(* CODESYS project ers_co2_payload_decoder.library
   Company: PXL-Tech
   Title: ERS_CO2 Payload Decoder
   Placeholder: ERS_CO2 Payload Decoder
   Version: 1.0

Project tree, tasks and I/O mapping:
  libraries: Tc2_Standard, * (Beckhoff Automation GmbH); Tc2_System, * (Beckhoff Automation GmbH); Tc2_Utilities, * (Beckhoff Automation GmbH); Tc3_Module, * (Beckhoff Automation GmbH)
  DUTs/
  GVLs/
  POUs/
    function block ERS_CO2_PayloadDecoder [ST]
    program MAIN [ST]
  Version/
    global variables Global_Version
  VISUs/
*)

// Version/Global_Version
{attribute 'TcGenerated'}
// This function has been automatically generated from the project information.
VAR_GLOBAL CONSTANT
	{attribute 'const_non_replaced'}
	{attribute 'linkalways'}
	stLibVersion_ERS_CO2_Payload_Decoder : ST_LibVersion := (iMajor := 1, iMinor := 0, iBuild := 0, iRevision := 0, sVersion := '1.0');
END_VAR

// POUs/ERS_CO2_PayloadDecoder
FUNCTION_BLOCK ERS_CO2_PayloadDecoder
VAR_INPUT
	dataString 		: STRING(32);
END_VAR
VAR_OUTPUT
	Temperature 	: REAL;		//Temp -3276.8°C - 3276.7°C
	Humidity 		: BYTE;		//Humidity 0-100%
	X 				: REAL;		//Acceleration X -128 --> 127 +/-63 = 1G
	Y 				: REAL;		//Acceleration Y -128 --> 127 +/-63 = 1G
	Z 				: REAL;		//Acceleration Z -128 --> 127 +/-63 = 1G
	Light 			: WORD; 	//Light 0 - 65535 Lux
	Motion 			: BYTE;		//No of motion 0-255
	Co2				: WORD;		//Co2 0-65535 ppm 
	Vdd				: WORD;		//VDD 0-65535mV
	Analog1			: WORD;		//VDD 0-65535mV
	Lat				: DWORD;	//Latitude binary
	Lon				: DWORD;	//Longitude binary
	Pulse1			: WORD;		//Relative pulse count
	pulseAbs		: DWORD;	//no 0 - 0xFFFFFFFF
	ExternalTemp	: REAL;		//External temp -3276.5C-->3276.5C
	Digital			: BYTE;		//Value 1 or 0
	Distance		: WORD;		//Distance in mm
	AccMotion		: BYTE;		//Number of vibration/motion
	IrInternalTemp	: REAL;		//Internal temp -3276.5C - 3276.5C
	IrExternalTemp	: REAL;		//External temp -3276.5C - 3276.5C
	Occupancy		: BYTE;		//Data
	Waterleak		: BYTE;		//Data 0-255
	Pressure		: REAL;		//Pressure data(hPa)
	SoundPeak		: BYTE;		//Sound peak
	SoundAvg		: BYTE;		//Sound average
	Pulse2			: WORD;		//0 - 0xFFFF
	PulseAbs2		: DWORD;	//no 0 - 0xFFFFFFFF
	Analog2			: WORD;		//Voltage in mV
	ExternalTemp2	: REAL;		//External temp2 -3276.5C - 3276.5C
	
	msgIDs			: ARRAY[1..8] OF BYTE;
END_VAR
VAR
	dataBuf			: ARRAY[1..16] OF BYTE;
	i				: INT;
	j				: INT;
END_VAR
VAR CONSTANT
	ID_Temp			:	BYTE	:= 16#01;	//Temperature
	ID_Rh			:	BYTE	:= 16#02;	//Humidity
	ID_Acc			:	BYTE	:= 16#03;	//X, Y, Z
	ID_Light		:	BYTE	:= 16#04;	//Light
	ID_Motion		:	BYTE	:= 16#05;	//Motion
	ID_Co2			:	BYTE	:= 16#06;	//Co2
	ID_Vdd			:	BYTE	:= 16#07;	//Vdd
	ID_Analog1		:	BYTE	:= 16#08;	//Analog1
	ID_Gps			:	BYTE	:= 16#09;	//Lat, Lon
	ID_Pulse1		:	BYTE	:= 16#0A;	//Pulse1
	ID_Pulse1_Abs	:	BYTE	:= 16#0B;	//Pulse1_Abs
	ID_Ext_Temp1	:	BYTE	:= 16#0C;	//ExternalTemp
	ID_Ext_Digital	:	BYTE	:= 16#0D;	//Digital
	ID_Ext_distance	:	BYTE	:= 16#0E;	//Distance
	ID_Acc_Motion	:	BYTE	:= 16#0F;	//AccMotion
	ID_Ir_Temp		:	BYTE	:= 16#10;	//IrInternalTemp, IrExternalTemp
	ID_Occupancy	:	BYTE	:= 16#11;	//Occupancy
	ID_Waterleak	:	BYTE	:= 16#12;	//Waterleak
	ID_Grideye		:	BYTE	:= 16#13;
	ID_Pressure		:	BYTE	:= 16#14;	//Pressure
	ID_Sound		:	BYTE	:= 16#15;	//SoundPeak, SoundAvg
	ID_Pulse2		:	BYTE	:= 16#16;	//Pulse2
	ID_Pulse2_Abs	:	BYTE	:= 16#17;	//Pulse2_Abs
	ID_Analog2		:	BYTE	:= 16#18;	//Analog2
	ID_Ext_Temp2	:	BYTE	:= 16#19;	//ExternalTemp2
END_VAR

HEXSTR_TO_DATA(dataString, ADR(dataBuf), SIZEOF(dataBuf));

j := 1;
MEMSET(ADR(msgIDs), 0, SIZEOF(msgIDs));

FOR i := 1 TO 15 BY 1 DO;
	CASE dataBuf[i] OF
		ID_Temp:
			Temperature := WORD_TO_REAL(SHL(dataBuf[i + 1], 8) OR dataBuf[i + 2]) / 10;
			msgIDs[j] := ID_Temp;
			j := j + 1;
			i := i + 2;
		ID_Rh:
			Humidity := dataBuf[i + 1];
			msgIDs[j] := ID_Rh;
			j := j + 1;
			i := i + 1;
		ID_Acc:
			X := dataBuf[i + 1];
			Y := dataBuf[i + 2];
			Z := dataBuf[i + 3];
			msgIDs[j] := ID_Acc;
			j := j + 1;
			i := i + 3;
		ID_Light:
			Light := SHL(dataBuf[i + 1], 8) OR dataBuf[i + 2];
			msgIDs[j] := ID_Light;
			j := j + 1;
			i := i + 2;
		ID_Motion:
			Motion := dataBuf[i + 1];
			msgIDs[j] := ID_Motion;
			j := j + 1;
			i := i + 1;
		ID_Co2:
			Co2 := SHL(dataBuf[i + 1], 8) OR dataBuf[i + 2];
			msgIDs[j] := ID_Co2;
			j := j + 1;
			i := i + 2;
		ID_Vdd:
			Vdd := SHL(dataBuf[i + 1], 8) OR dataBuf[i + 2];
			msgIDs[j] := ID_Vdd;
			j := j + 1;
			i := i + 2;
		ID_Analog1:
			Analog1 := SHL(dataBuf[i + 1], 8) OR dataBuf[i + 2];
			msgIDs[j] := ID_Analog1;
			j := j + 1;
			i := i + 2;
		ID_Gps:
			Lat := SHL(dataBuf[i + 1], 16) OR SHL(dataBuf[i + 2], 8) OR dataBuf[i + 3];
			Lon := SHL(dataBuf[i + 4], 16) OR SHL(dataBuf[i + 5], 8) OR dataBuf[i + 6];
			msgIDs[j] := ID_Gps;
			j := j + 1;
			i := i + 6;
		ID_Pulse1:
			Pulse1 := SHL(dataBuf[i + 1], 8) OR dataBuf[i + 2];
			msgIDs[j] := ID_Pulse1;
			j := j + 1;
			i := i + 2;
		ID_Pulse1_Abs:
			PulseAbs := SHL(dataBuf[i + 1], 24) OR SHL(dataBuf[i + 2], 16) OR  SHL(dataBuf[i + 3], 8) OR dataBuf[i + 4];
			msgIDs[j] := ID_Pulse1_Abs;
			j := j + 1;
			i := i + 4;
		ID_Ext_Temp1:
			ExternalTemp := WORD_TO_REAL(SHL(dataBuf[i + 1], 8) OR dataBuf[i + 2]) / 10;
			msgIDs[j] := ID_Ext_Temp1;
			j := j + 1;
			i := i + 2;
		ID_Ext_Digital:
			Digital := dataBuf[i + 1];
			msgIDs[j] := ID_Ext_Digital;
			j := j + 1;
			i := i + 1;
		ID_Ext_distance:
			Distance := SHL(dataBuf[i + 1], 8) OR dataBuf[i + 2];
			msgIDs[j] := ID_Ext_distance;
			j := j + 1;
			i := i + 2;
		ID_Acc_Motion:
			AccMotion := dataBuf[i + 1];
			msgIDs[j] := ID_Acc_Motion;
			j := j + 1;
			i := i + 1;
		ID_Ir_Temp:
			IrInternalTemp := WORD_TO_REAL(SHL(dataBuf[i + 1], 8) OR dataBuf[i + 2]) / 10;
			IrExternalTemp := WORD_TO_REAL(SHL(dataBuf[i + 3], 8) OR dataBuf[i + 4]) / 10;
			msgIDs[j] := ID_Ir_Temp;
			j := j + 1;
			i := i + 4;
		ID_Occupancy:
			Occupancy := dataBuf[i + 1];
			msgIDs[j] := ID_Occupancy;
			j := j + 1;
			i := i + 1;
		ID_Waterleak:
			Waterleak := dataBuf[i + 1];
			msgIDs[j] := ID_Waterleak;
			j := j + 1;
			i := i + 1;
		ID_Grideye:
			msgIDs[j] := ID_Grideye;
			j := j + 1;
			i := i + 65;
		ID_Pressure:
			Pressure := DWORD_TO_REAL(SHL(dataBuf[i + 1], 24) OR SHL(dataBuf[i + 2], 16) OR  SHL(dataBuf[i + 3], 8) OR dataBuf[i + 4]) / 1000;
			msgIDs[j] := ID_Pressure;
			j := j + 1;
			i := i + 4;
		ID_Sound:
			SoundPeak := dataBuf[i + 1];
			SoundAvg := dataBuf[i + 2];
			msgIDs[j] := ID_Sound;
			j := j + 1;
			i := i + 2;
		ID_Pulse2:
			Pulse2 := SHL(dataBuf[i + 1], 8) OR dataBuf[i + 2];
			msgIDs[j] := ID_Pulse2;
			j := j + 1;
			i := i + 2;
		ID_Pulse2_Abs:
			PulseAbs2 := SHL(dataBuf[i + 1], 24) OR SHL(dataBuf[i + 2], 16) OR  SHL(dataBuf[i + 3], 8) OR dataBuf[i + 4];
			msgIDs[j] := ID_Pulse2_Abs;
			j := j + 1;
			i := i + 4;
		ID_Analog2:
			Analog2  := SHL(dataBuf[i + 1], 8) OR dataBuf[i + 2];
			msgIDs[j] := ID_Analog2;
			j := j + 1;
			i := i + 2;
		ID_Ext_Temp2:
			ExternalTemp2  := WORD_TO_REAL(SHL(dataBuf[i + 1], 8) OR dataBuf[i + 2]) / 10;
			msgIDs[j] := ID_Ext_Temp2;
			j := j + 1;
			i := i + 2;
		ELSE
			i := 16;
	 END_CASE
END_FOR

END_FUNCTION_BLOCK

// POUs/MAIN
PROGRAM MAIN
VAR
	fb_Decoder : ERS_CO2_PayloadDecoder;
	dataStr :STRING(32) := '0100e202290400270506060308070d62';
END_VAR

fb_Decoder(dataString := dataStr);
;

END_PROGRAM
